{attribute 'GeneratedUsingTerminal: EL3423-0000-0020'}
{attribute addProperty BoxType "EL3423-0000-0020"}
{attribute addProperty Id "TxPDO_ToggleAT %I*BOOL1Active_EnergyAT %I*REAL4Apparent_EnergyAT %I*REAL4Reactive_EnergyAT %I*REAL4"}
{attribute addProperty CRC "2963328472"}
{attribute addProperty Size "13"}
TYPE Total_Interval_Energy_Reduced_B0A0CDD8 :
STRUCT
	{attribute addProperty Name "TxPDO_Toggle"}
	TxPDO_Toggle AT %I* : BOOL;
	{attribute addProperty Name "Active_Energy"}
	Active_Energy AT %I* : REAL;
	{attribute addProperty Name "Apparent_Energy"}
	Apparent_Energy AT %I* : REAL;
	{attribute addProperty Name "Reactive_Energy"}
	Reactive_Energy AT %I* : REAL;
END_STRUCT
END_TYPE

(* stored: Version 1.2.0.0, ProductVersion 3.1.4024.9
   DUT Total_Interval_Energy_Reduced_B0A0CDD8: Id {1f20924b-d3d2-481d-99e0-e18803079dc7} *)
